Fanuc KAREL source: polygon.klc

PROGRAM class_name
%NOBUSYLAMP
%COMMENT = 'polygon object'
%NOLOCKGROUP

--*** ..todo:: Does not work for polygons with holes

%include namespace.m

%include errors.klt
%include systemvars.klt
%include systemlib.types.klt
%include pathlib.c.klt
%include pathlib.t.klt
%include draw.klt

VAR
  canvas : PATH nodedata = t_VERTEX
  sub_poly : PATH nodedata = t_VERTEX
  -- ..Note:: `sub_poly` maybe should be a seperate type without
  --          nextPoly, prevPoly, polygon, and include holes member list
  hull : PATH nodedata = t_VERTEX

  lines : PATH nodedata = t_SEG2D_POLY
  contours : PATH nodedata = t_VEC_PATH
  fl : FILE
  origin : XYZWPR
  params : t_RASTER
  -- toggle if you want to raster lines on the boundary of the shape
  -- if false it will exclude the boundary
  rast_bounds : BOOLEAN

  -- ..Note:: centroids are calculated in bounding box calculations
  --          check that bounding boxes are calculated per polygon,
  --          not whole drawing

%from systemlib.klh %import VEC, VEC2D
%from strings.klh %import s_to_vec
%from math.klh %import arclength, arcangle, norm, rotz
%from pose.klh %import vector_to_pose
%include csv.klh
%include errors.klh
%include draw.klh

%include polygon.klh
%include polygon.private.klh


-- ** private **

ROUTINE clear_hull
  VAR
    i : INTEGER
    status : INTEGER
  BEGIN
    i = PATH_LEN(hull)
    WHILE PATH_LEN(hull) > 0 DO
		  DELETE_NODE(hull,i,status)
      CHK_STAT(status)
      i = i - 1
	  ENDWHILE
  END clear_hull

ROUTINE clear_poly
  VAR
    i : INTEGER
    status : INTEGER
  BEGIN
    i = PATH_LEN(p)
    WHILE PATH_LEN(p) > 0 DO
		  DELETE_NODE(p,i,status)
      CHK_STAT(status)
      i = i - 1
	  ENDWHILE
  END clear_poly

ROUTINE clear_lines
  VAR
    i : INTEGER
    status : INTEGER
  BEGIN
    i = PATH_LEN(lines)
    WHILE PATH_LEN(lines) > 0 DO
		  DELETE_NODE(lines,i,status)
      CHK_STAT(status)
      i = i - 1
	  ENDWHILE
  END clear_lines

ROUTINE clear_contours
  VAR
    i : INTEGER
    status : INTEGER
  BEGIN
    i = PATH_LEN(contours)
    WHILE PATH_LEN(contours) > 0 DO
		  DELETE_NODE(contours,i,status)
      CHK_STAT(status)
      i = i - 1
	  ENDWHILE
  END clear_contours

ROUTINE new_sub_poly
  VAR
    nde_strt, nde_end : INTEGER
    i : INTEGER
    status : INTEGER
    idx : VECTOR2Di
  BEGIN
    nde_strt = 1; nde_end = PATH_LEN(canvas);
    --find polygon
    IF (polygon > 0) THEN
      i = 1
      REPEAT
        nde_strt = i
        --handle uninitialized nextPoly
        IF UNINIT(canvas[i].nextPoly) THEN
          nde_end = PATH_LEN(canvas)
        ELSE
          nde_end = canvas[i].nextPoly - 1
        ENDIF

        i = canvas[i].nextPoly
      UNTIL(canvas[i].polygon > polygon)
    ENDIF

    --clear to sub path
    clear_poly(sub_poly)
    COPY_PATH(canvas, nde_strt, nde_end, sub_poly, status)
    CHK_STAT(status)

    idx.x = nde_strt
    idx.y = nde_end

    RETURN(idx)

  END new_sub_poly

ROUTINE update_last_poly
  VAR
    i : INTEGER
    polygon : INTEGER
  BEGIN
    --append pointer to next polygon if other
    --polygons exist
    i = PATH_LEN(canvas)
    IF i > 0 THEN
      IF NOT UNINIT(canvas[i].polygon) THEN
        polygon = canvas[i].polygon + 1
      ELSE
        polygon = 1
      ENDIF

      WHILE (i > 0) DO
        IF UNINIT(canvas[i].nextPoly) THEN
          canvas[i].nextPoly = PATH_LEN(canvas) + 1
        ENDIF
        i = i - 1
      ENDWHILE
    ELSE
      polygon = 1
    ENDIF

    RETURN(polygon)
  END update_last_poly

-- ** public **

ROUTINE delete
  VAR
    i : INTEGER
    status : INTEGER
  BEGIN
    i = PATH_LEN(canvas)
    WHILE PATH_LEN(canvas) > 0 DO
		  DELETE_NODE(canvas,i,status)
      i = i - 1
	  ENDWHILE
    --uninitialize the canvas
    SET_UNINIT_F('class_name', 'origin')

    rast_bounds = FALSE

    --clear hull
    clear_hull
    --clear to sub path
    clear_poly(sub_poly)

    clear_lines
    clear_contours
  END delete

ROUTINE new
%define DEFAULT_PITCH 3
  BEGIN
    delete
    set_canvas((ZEROPOS(1)))
    rast_bounds = TRUE

    --set default params
    params.start_angle = 0
    params.line_width = 0
    params.line_pitch = DEFAULT_PITCH
    params.dir = 1
    params.wall_lines = 0
  END new

ROUTINE init
  BEGIN
    delete
    set_canvas(frm_)
    rast_bounds = boundary

    --fill params
    params.start_angle = start_angle_
    params.dir = dir_
    params.wall_lines = wall_lines_
    params.line_width = line_width_
    params.line_pitch = line_pitch_
  END init

ROUTINE init2
  BEGIN
    delete
    set_canvas(frm_)
    rast_bounds = boundary

    --fill params
    params.start_angle = rast.start_angle
    params.dir = rast.dir
    params.wall_lines = rast.wall_lines
    params.line_width = rast.line_width
    params.line_pitch = rast.line_pitch
  END init2

--clear the canvas, but keep the canvas
ROUTINE erase
  BEGIN
    --clear drawing
    clear_poly(canvas)
    clear_poly(sub_poly)

    --clear hull
    clear_hull

    --clear rasters
    clear_lines
    clear_contours
  END erase

ROUTINE import_shape
  VAR
    header : STRING[16]
    str : STRING[32]
    b : BOOLEAN
    v : VECTOR
    vert : INTEGER
    poly : INTEGER
    status : INTEGER
  BEGIN
    csv__read_open(filename, fl)
    --read header
    header = csv__read_line(filename, fl)

    clear_poly(sub_poly)
    --vertex count
    vert = 0
    --intialize polygon count
    poly = 1
    REPEAT
      vert = vert + 1

      --read line
      b = csv__read_line_ref(filename, fl, str)

      IF b THEN
        --put string into vector
        v = s_to_vec(str, ',')

        IF TRUNC(v.z) > poly THEN
          --append previous polygon into canvas (canvas)
          append_polygon(sub_poly)
          clear_poly(sub_poly)

          --add first vertex of next polygon
          poly = TRUNC(v.z)
          APPEND_NODE(sub_poly,status)
          sub_poly[PATH_LEN(sub_poly)].coords = VEC2D(v.x, v.y)
          sub_poly[PATH_LEN(sub_poly)].polygon = poly
        ELSE
          --add vertex
          APPEND_NODE(sub_poly,status)
          sub_poly[PATH_LEN(sub_poly)].coords = VEC2D(v.x, v.y)
          sub_poly[PATH_LEN(sub_poly)].polygon = poly
        ENDIF
      ELSE
        --end of file append polygon into canvas (canvas)
        append_polygon(sub_poly)
        clear_poly(sub_poly)
      ENDIF
    UNTIL(NOT b)

    csv__read_close(fl)

  END import_shape

ROUTINE set_canvas
  BEGIN
    origin = frm_
  END set_canvas

ROUTINE flip_canvas
  VAR
    bbox : t_RECT
    len : REAL
  BEGIN
    --get length of the drawing, and translate by that length
    len = get_canvas_length
    origin = origin:POS(0,0,len,0,180,0,(ZEROPOS(1).config_data))
  END flip_canvas

ROUTINE raster_on_boundary
  BEGIN
    rast_bounds = boundary
  END raster_on_boundary

ROUTINE set_params
  BEGIN
    params.start_angle = start_angle
    params.dir = dir
    params.wall_lines = wall_lines
    params.line_width = line_width
    params.line_pitch = line_pitch
  END set_params

ROUTINE get_params
  BEGIN
    RETURN(params)
  END get_params

ROUTINE append_vertex
  VAR
    status : INTEGER
    nd : t_VERTEX
  BEGIN
    IF UNINIT(origin) THEN
      karelError(VAR_UNINIT,'class_name member "origin" needs to' + &
                ' be set before building polygons', ER_ABORT)
    ENDIF
    APPEND_NODE(canvas,status)
    CHK_STAT(status)
    nd.coords = VEC2D(vertex.x, vertex.y)
    nd.polygon = polygon
    canvas[PATH_LEN(canvas)] = nd
  END append_vertex

ROUTINE append_polygon
  VAR
    i : INTEGER
    polygon : INTEGER
    lastPoly : INTEGER
  BEGIN
    polygon = update_last_poly

    --retain last index to point to prevPoly
    IF PATH_LEN(canvas) > 0 THEN lastPoly = PATH_LEN(canvas); ENDIF

    FOR i=1 TO PATH_LEN(verticies) DO
      append_vertex(verticies[i].coords, (polygon))
      IF NOT UNINIT(lastPoly) AND (lastPoly > 0) THEN
        canvas[PATH_LEN(canvas)].prevPoly = lastPoly
      ENDIF
    ENDFOR
  END append_polygon

ROUTINE append_polygon_array
  VAR
    i : INTEGER
    polygon : INTEGER
    lastPoly : INTEGER
  BEGIN
    polygon = update_last_poly

    --retain last index to point to prevPoly
    IF PATH_LEN(canvas) > 0 THEN lastPoly = PATH_LEN(canvas); ENDIF

    FOR i=1 TO ARRAY_LEN(verticies) DO
      append_vertex(verticies[i], (polygon))
      IF NOT UNINIT(lastPoly) THEN
        canvas[PATH_LEN(canvas)].prevPoly = lastPoly
      ENDIF
    ENDFOR
  END append_polygon_array

ROUTINE get_poly
  VAR
    i, nd, status : INTEGER
  BEGIN
    IF polygon = 0 THEN
      COPY_PATH(canvas, 1, PATH_LEN(canvas), out_poly, status)
      CHK_STAT(status)
    ELSE
      nd = 1
      REPEAT
        i = nd
        IF UNINIT(canvas[i].nextPoly) THEN
          nd = PATH_LEN(canvas)
        ELSE
          nd = canvas[i].nextPoly
        ENDIF
      UNTIL(canvas[i].polygon = polygon)

      COPY_PATH(canvas, 1, nd, out_poly, status)
      CHK_STAT(status)
    ENDIF
  END get_poly

ROUTINE get_lines
  VAR
    status : INTEGER
  BEGIN
    COPY_PATH(lines, start_i, end_i, out_lines, status)
    CHK_STAT(status)
  END get_lines

ROUTINE get_contours
  VAR
    status : INTEGER
  BEGIN
    COPY_PATH(contours, start_i, end_i, out_cntrs, status)
    CHK_STAT(status)
  END get_contours

ROUTINE get_bounding_box_drawing
  VAR
    bbox : t_RECT
  BEGIN
    bbox = draw__bounding_box(canvas, (params.start_angle))
    --convert to world coordinates
    RETURN(bbox)
  END get_bounding_box_drawing

ROUTINE get_bounding_box_poly
  VAR
    bbox : t_RECT
    idx : VECTOR2Di
  BEGIN
    --get individual polygon and store in `sub_poly`
    idx = new_sub_poly(polygon)
    bbox = draw__bounding_box(sub_poly, (params.start_angle))
    --convert to world coordinates
    RETURN(bbox)
  END get_bounding_box_poly

ROUTINE get_canvas_length
  VAR
    bbox : t_RECT
  BEGIN
    --get bounding box
    bbox = get_bounding_box_drawing

    -- get length of bounding box along its longitude
    RETURN(math__norm(bbox.verts[4]-bbox.verts[1]))
  END get_canvas_length

ROUTINE get_polygon_count
  BEGIN
    RETURN(canvas[PATH_LEN(canvas)].polygon)
  END get_polygon_count

ROUTINE translate_canvas
  BEGIN
    origin = origin:POS(vec.x,vec.y,vec.z,0,0,0,(ZEROPOS(1).config_data))
  END translate_canvas

ROUTINE rotate_polygon
  VAR
    i, j : INTEGER
    p : XYZWPR
    center : VECTOR
    idx : VECTOR2Di
  BEGIN
    --get isolated polygon and calculate center point
    idx = new_sub_poly(polygon)
    --get center
    center = draw__psuedo_center(sub_poly)

    --use for updating canvas
    j = idx.x
    FOR i=1 TO PATH_LEN(sub_poly) DO
      --put vertex in object (polygon) space
      p = pose__vector_to_pose((sub_poly[i].coords - center), VEC(0,0,0), (ZEROPOS(1).config_data))
      --rotate vertex
      p = math__rotz(p, angle)
      --put back into vector and into canvas space
      sub_poly[i].coords = VEC(p.x, p.y, p.z) + center
      --copy back into canvas
      canvas[j].coords = sub_poly[i].coords

      j = j + 1
    ENDFOR

  END rotate_polygon

ROUTINE scale_polygon_along_axes
  --factor should be between in mm for the x and y axis.
  --will calculate the distance to each axis and scale
  --down to that axis depending on the fraction.
  VAR
    i, j : INTEGER
    v : VECTOR
    center : VECTOR
    tang_vec, perp_vec : VECTOR
    amt : REAL
    idx : VECTOR2Di
  BEGIN
    -- ..Note:: `params.start_angle` must be set before running canvas
    --           function

    --get isolated polygon
      -- ..Note:: do not use `get_bounding_box_poly` as you need
      --          to save idx to update `canvas` as well as `sub_poly`
    idx = new_sub_poly(polygon)
    --get center
    center = draw__psuedo_center(sub_poly)

    --scale along the raster angle
      --x-axis vector
    tang_vec = draw__angle_to_vector(params.start_angle)
    tang_vec = tang_vec/math__norm(tang_vec)
      --y-axis vector
    perp_vec = draw__angle_to_vector(params.start_angle + 90)
    perp_vec = perp_vec/math__norm(perp_vec)

    --use for updating canvas
    j = idx.x
    FOR i=1 TO PATH_LEN(sub_poly) DO
      --put vertex in object (polygon) space
      v = (sub_poly[i].coords - center)
      --x-axis
       --determine above or below axis
      IF (v@tang_vec > 0) THEN
        -- move in positive direction
        v.x = factor.x+v.x
        --do not cross axis
        IF v.x < 0 THEN v.x = 0 ; ENDIF
      ELSE
        -- move in negative direction
        v.x = -1*factor.x+v.x
        --do not cross axis
        IF v.x > 0 THEN v.x = 0 ; ENDIF
      ENDIF

      --y-axis
       --determine above or below axis
      IF (v@perp_vec > 0) THEN
        -- move in positive direction
        v.y = factor.y+v.y
        --do not cross axis
        IF v.y < 0 THEN v.y = 0 ; ENDIF
      ELSE
        -- move in negative direction
        v.y = -1*factor.y+v.y
        --do not cross axis
        IF v.y > 0 THEN v.y = 0 ; ENDIF
      ENDIF

      --put back into vector and into canvas space
      sub_poly[i].coords = v + center
      --copy back into canvas
      canvas[j].coords = sub_poly[i].coords

      j = j + 1
    ENDFOR

  END scale_polygon_along_axes

ROUTINE trace
  VAR
    i : INTEGER
  BEGIN
    --clear previous contours
    clear_contours

    --get walls
    i = 0
    WHILE (i < params.wall_lines) DO
      --clear inset
      clear_poly(sub_poly)
      --inset by width of line to fill within boundaries
      --inset and trace each polygon on the canvas
       -- **fix** :: currently insetting over full list. Shouldn't it be the sub polygon
       --            might have to add extra t_VERTEX memeber to store result
      draw__inset_polygon(canvas, (params.line_width/2 + i*params.line_pitch), hull, sub_poly)
      --trace polygon
      draw__trace(sub_poly, params.start_angle, (params.dir), line_type, contours)
      draw__calc_tangent_segment(contours)
      i = i + 1
    ENDWHILE

  END trace

ROUTINE raster
  VAR
    i, status : INTEGER
  BEGIN
    clear_lines
    --trace contours if wall_lines > 0
    trace(line_type)
    --raster the interior over whole canvas
    draw__raster_lines(canvas, hull, params.start_angle, params.line_width, params.line_pitch, (params.dir), rast_bounds, lines)

  END raster

ROUTINE lines_to_vec_path
  VAR
    i : INTEGER
    status : INTEGER
    prev_vert, curr_vert, next_vert : INTEGER
  BEGIN
    IF UNINIT(origin) THEN
      karelError(VAR_UNINIT,'class_name member "origin" needs to' + &
                ' be set before converting', ER_ABORT)
    ENDIF

    --convert lines
    FOR i=1 TO PATH_LEN(lines) DO
      --r0
      APPEND_NODE(out_lines, status)
      out_lines[PATH_LEN(out_lines)].v = origin:lines[i].r0
      out_lines[PATH_LEN(out_lines)].code = PTH_MOVETO
      out_lines[PATH_LEN(out_lines)].polygon = lines[i].polygon
      out_lines[PATH_LEN(out_lines)].tangent = origin:lines[i].tangent

      --r1
      APPEND_NODE(out_lines, status)
      out_lines[PATH_LEN(out_lines)].v = origin:lines[i].r1
      out_lines[PATH_LEN(out_lines)].code = PTH_CLOSE
      out_lines[PATH_LEN(out_lines)].polygon = lines[i].polygon
      out_lines[PATH_LEN(out_lines)].tangent = origin:lines[i].tangent
    ENDFOR
  END lines_to_vec_path

ROUTINE contours_to_vec_path
  VAR
    i, status : INTEGER
    next_vert,prev_vert : INTEGER
  BEGIN
    IF UNINIT(origin) THEN
      karelError(VAR_UNINIT,'class_name member "origin" needs to' + &
                ' be set before converting', ER_ABORT)
    ENDIF

    --convert contours
    FOR i=1 TO PATH_LEN(contours) DO
      APPEND_NODE(out_cntrs, status)
      out_cntrs[PATH_LEN(out_cntrs)].v = origin:contours[i].v
      out_cntrs[PATH_LEN(out_cntrs)].code = contours[i].code
      out_cntrs[PATH_LEN(out_cntrs)].polygon = contours[i].polygon
      out_cntrs[PATH_LEN(out_cntrs)].tangent = origin:contours[i].tangent
    ENDFOR

  END contours_to_vec_path

  BEGIN
  END class_name
